TYPE DUT_HMI_EV_Info :
STRUCT
	Enable	 : BOOL;
	dTime 	 : UINT;
	Error 	 : BOOL;	
END_STRUCT
END_TYPE

(* stored: Version 1.1.0.1, ProductVersion 3.1.4024.15
   DUT DUT_HMI_EV_Info: Id {5aec27aa-4fbb-4dc9-9d41-2140b9beb64d} *)
